FUNCTION_BLOCK IndexMover EXTENDS FB_Mover
VAR_INPUT
	TrackState : E_Xts_StateMachine;
	XtsTrack : IXtsTrack;
END_VAR
VAR_OUTPUT
END_VAR
VAR
	moverSequence : IndexMoverSequence;
END_VAR
VAR_IN_OUT
	StationArray : ARRAY[*] OF IStation;
END_VAR

SUPER^();

moverSequence(ThisMover	 := THIS^, XtsTrack := XtsTrack);

END_FUNCTION_BLOCK

(* stored: Version 1.1.0.1, ProductVersion 3.1.4024.9
   POU IndexMover: Id {4b45940e-4817-4260-a891-e07dd3ca95d8}, SpecialFunc None *)
